# EPICS autosave request: linkamT96App/Db/Linkam_settings.req
$(P):CONFIG.SCAN
$(P):STATUS.SCAN
$(P):STAGE:CONFIG.SCAN
$(P):TEMP.SCAN
$(P):DISABLE.VAL
$(P):DSC.SCAN
$(P):STARTHEAT.VAL
$(P):RAMPRATE:SET.VAL
$(P):RAMPRATE.SCAN
$(P):HOLDTIME:SET.VAL
$(P):HOLDTIME.SCAN
$(P):SETPOINT:SET.VAL
$(P):SETPOINT.SCAN
$(P):POWER.SCAN
$(P):LNP_SPEED:SET.VAL
$(P):LNP_SPEED.SCAN
$(P):LNP_MODE:SET.VAL
